PROGRAM PRG_LVCP5_Group6
VAR
    // Function Block Instance
    fbContactor: FB_ContactorControl;

    // Contactor 1 IO Structure  
    stContactor_IO: ST_ContactorIO;
    
    // Başlangıç konfigürasyonu için flag
    bContactorInitDone: BOOL := FALSE;
    bCapacitorInitDone: BOOL := FALSE;	
END_VAR



	M_Contactor();
	
	M_Capacitor();

METHOD M_Capacitor : BOOL
VAR
    nGroupIndex : INT;
END_VAR

nGroupIndex := 5;  // Grup 6 için index

IF NOT bCapacitorInitDone THEN
    // Grup 6 değerlerini ata
    GVL_LVCP5.astCompensationGroups[nGroupIndex].rPower := 25.0;
    GVL_LVCP5.astCompensationGroups[nGroupIndex].rVoltage := 450.0;
    GVL_LVCP5.astCompensationGroups[nGroupIndex].nQuantity := 2;
    GVL_LVCP5.astCompensationGroups[nGroupIndex].sTagPrefix := '+EP8-31C1';
    GVL_LVCP5.astCompensationGroups[nGroupIndex].sProductCode := 'ENT.CXD-450-10';
    
    bCapacitorInitDone := TRUE;
END_IF

// Grup 6 aktif durumu
GVL_LVCP5.abGroupActive[nGroupIndex] := stContactor_IO.bFeedback;

M_Capacitor := TRUE;
END_METHOD

METHOD M_Contactor : BOOL
VAR_INPUT
END_VAR
IF NOT bContactorInitDone THEN
    // Konfigürasyon parametreleri
    GVL_LVCP5.stGroup6_ContactorHMI.stConfig.sProjectCode := '+EP8-32K1';
    GVL_LVCP5.stGroup6_ContactorHMI.stConfig.sProductCode := 'SCH LC1D40A3P7';
    GVL_LVCP5.stGroup6_ContactorHMI.stConfig.rRatedCurrent := 40.0;
    GVL_LVCP5.stGroup6_ContactorHMI.stConfig.rRatedVoltage := 690.0;
    GVL_LVCP5.stGroup6_ContactorHMI.stConfig.nPhaseCount := 3;
    GVL_LVCP5.stGroup6_ContactorHMI.stConfig.tFeedbackDelay := T#500MS;
    GVL_LVCP5.stGroup6_ContactorHMI.stConfig.tWeldedDelay := T#2S;
    GVL_LVCP5.stGroup6_ContactorHMI.stConfig.dwOperationLimit := 100000;
    
    // Başlangıç bakım sayacı
    GVL_LVCP5.stGroup6_ContactorHMI.stStatistics.dwRemainingOperations := GVL_LVCP5.stGroup6_ContactorHMI.stConfig.dwOperationLimit;
    
    bContactorInitDone := TRUE;
END_IF

// Function Block Çağrısı
fbContactor(
    // Fiziksel Girişler
    bFeedback 		:= stContactor_IO.bFeedback,
    bPLCControl 	:= stContactor_IO.bPLCControl,
    
    // Güvenlik Girişleri
    bSafetyLoop 	:= GVL_Alarm.bSafetyLoop,
    bInterlock 		:= FALSE,
    
    // Sistem Girişleri
    bMasterReset 	:= GVL_Alarm.bMasterReset,
    
    // HMI Bağlantısı
    stHMI 			:= GVL_LVCP5.stGroup6_ContactorHMI,
    
    // Fiziksel Çıkış
    bOutput 		=> stContactor_IO.bOutput
);

M_Contactor := TRUE;
END_METHOD

END_PROGRAM

(* stored: Version 1.1.0.1, ProductVersion 3.1.4024.15
   POU PRG_LVCP5_Group6: Id {d9791c99-1725-48b1-b5f1-b2f3fa1526d6}, SpecialFunc None
   Method M_Capacitor: Id {2eb0d13a-378c-45ae-8f52-a8dc35e1b2a2}
   Method M_Contactor: Id {cb83056e-2132-4d4a-a25f-decfbe55b048} *)
